ABB RobotStudio station: Obelix2_20190304-113324.rsstn

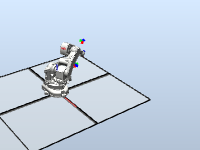
Station Obelix2 (saved by RobotStudio 6.8.8148.134)
Controller IRB_140T_6kg_0.81m
  mechanical unit ROB_1: IRB140T_6_81_C_03, 6 joints, base frame (0, 0, 0) mm
Layout (positions relative to the parent item):
  - IRB140T_6_81_C_03 [mechanism, from Robots\IRB140T_6_81_C_G_03.rslib] at (0, 0, 0) mm; joint values [1.9862, 0.8146, -0.2687, 3.1416, 0.4317, -3.1416] (rad or m)
  - conveyor [part]
  - ManipulationTable [part]
  - conveyor_2 [part]
  - Oven_2 [part]
Targets, tools, work objects and paths stored in the station, written as RAPID:
! task T_ROB1
MODULE ObelixMov
  CONST robtarget pHome:=[[507.9,-6.43,715.02],[0.697685,-0.00154316,0.716328,-0.0103435],[-1,-1,-1,0],[9E+09,9E+09,9E+09,9E+09,9E+09,9E+09]];
  CONST robtarget pOvenRef:=[[-291.029880742,659.908842444,594.297264732],[0.363486279,-0.625201176,0.407577419,0.55756781],[1,0,-1,0],[9E+09,9E+09,9E+09,9E+09,9E+09,9E+09]];
  PROC main()
    MoveJ pHome,v1000,fine,tool0;
    MoveJ pHome,v1000,fine,tool0;
  ENDPROC
ENDMODULE

